FUNCTION_BLOCK fbLightControl
		
VAR_INPUT
	bButton				: BOOL;
	bForceOff			: BOOL;
	bForceOn			: BOOL;

END_VAR
VAR_OUTPUT
	bLight				: BOOL;
	
END_VAR
VAR
	InputTrigger		: R_trig; 

	
END_VAR

// This is the first version, ignoring all debounce timers and other issues 
// Base function is a to allow switching a light on and of and having a general reset and general on ( used for construcion)

InputTrigger(CLK :=  bButton);

IF InputTrigger.Q THEN
	
	bLight := NOT(bLight);

END_IF

// Deze functie zorgt voor alles aan/Uit Functionaliteit
IF bForceOff THEN
	bLight := FALSE;
END_IF

IF bForceOn THEN
	bLight := TRUE;
END_IF

(*function notes: long klick functionality not added, most likley this will be part of another function
This could be a dedicated filter function linked to these functions as needed
*)

END_FUNCTION_BLOCK

(* stored: Version 1.1.0.1, ProductVersion 3.1.4024.11
   POU fbLightControl: Id {7f5342f2-aa10-4900-98e2-28409aed465b}, SpecialFunc None *)
